FUNCTION_BLOCK FB_AxisWriteParams
VAR_INPUT
	bExecute: BOOL;
	bReset: BOOL;
	stConfig: ST_AxisParams;
	stHardware: ST_AxisHardware;
END_VAR
VAR_IN_OUT
	Axis: AXIS_REF;
END_VAR
VAR_OUTPUT
	bInitPreOp: BOOL;
	bDone: BOOL;
	bBusy: BOOL;
	bError: BOOL;
	nErrorID: UDINT;
END_VAR
VAR
	bDoWrite: BOOL;
	fbNCWrite: FB_AxisWriteNC;
	fbCoEWrite: FB_AxisWriteCoE;
	fbPrepWrite: FB_AxisSetSlaveState;
	fbInitState: FB_AxisSetSlaveState;
	fbPreOpState: FB_AxisSetSlaveState;
END_VAR

// Do not write unless axis is disabled. Leave TRUE after done to avoid resetting errors, etc.
bDoWrite := bExecute AND (Axis.Status.MotionState = MC_AXISSTATE_DISABLED OR bDone);
// Move to PREOP to prepare for writing
fbPrepWrite(bExecute:=bDoWrite,
	stHardware:=stHardware,
	reqState:=EC_DEVICE_STATE_PREOP);
// The first time we're here, report that we've set to PREOP so master can move to OP
IF fbPrepWrite.bDone AND NOT fbPrepWrite.bError THEN
	bInitPreOP := TRUE;
END_IF
// Do the write
fbNCWrite(bExecute:=fbPrepWrite.bDone AND NOT fbPrepWrite.bError,
	bReset:=bReset,
	stConfig:=stConfig,
	Axis:=Axis);
fbCoEWrite(bExecute:=fbNCWrite.bExecute,
	bReset:=bReset,
	stHardware:=stHardware,
	stConfig:=stConfig,
	Axis:=Axis);
// Move to INIT and back to PRE-OP for params that need a full restart
fbInitState(bExecute:=fbNCWrite.bDone AND NOT fbNCWrite.bError AND NOT fbCoEWrite.bBusy AND NOT fbCoEWrite.bError,
	stHardware:=stHardware,
	reqState:=EC_DEVICE_STATE_INIT);
fbPreOpState(bExecute:=fbInitState.bDone AND NOT fbInitState.bError,
	stHardware:=stHardware,
	reqSTate:=EC_DEVICE_STATE_PREOP);
bDone := fbPreOpState.bDone;
bBusy := fbNCWrite.bBusy OR fbCoEWrite.bBusy OR fbPrepWrite.bBusy OR fbInitState.bBusy OR fbPreOpState.bBusy;
bError := fbNCWrite.bError OR fbCoEWrite.bError OR fbPrepWrite.bError OR fbInitState.bError OR fbPreOpState.bError;
IF fbNCWrite.nErrorID > 0 THEN
	nErrorID := fbNCWrite.nErrorID;
ELSIF fbCoeWrite.nErrorID > 0 THEN
	nErrorID := fbCoEWrite.nErrorID;
ELSIF fbPrepWrite.nErrId > 0 THEN
	nErrorID := fbPrepWrite.nErrId;
ELSIF fbInitSTate.nErrId > 0 THEN
	nErrorID := fbInitState.nErrId;
ELSE
	nErrorID := fbPreOpState.nErrId;
END_IF

END_FUNCTION_BLOCK

(* stored: Version 1.1.0.1, ProductVersion 3.1.4020.14
   POU FB_AxisWriteParams: Id {c12a06b7-df78-4119-aa24-9aeca1f8090f}, SpecialFunc None *)
